// TIA Portal project "Kap_5_Uebung_Schutztuer_CPU_1500_V14_V15.1" (V15.1)

(* hardware
DEVICE "S71500/ET200MP-Station_1"  S7-1500 station
   slot 0: "Profilschiene_0"  6ES7 590-1***0-0AA0
   slot 1: "PLC_1"  CPU 1511-1 PN  6ES7 511-1AK01-0AB0  V1.8
   slot 2: "AI 8xU/I/RTD/TC ST_1"  AI 8xU/I/RTD/TC ST  6ES7 531-7KF00-0AB0  V2.0
   slot 3: "AI 8xU/I/RTD/TC ST_2"  AI 8xU/I/RTD/TC ST  6ES7 531-7KF00-0AB0  V2.0
   slot 4: "AI 8xU/I/RTD/TC ST_3"  AI 8xU/I/RTD/TC ST  6ES7 531-7KF00-0AB0  V2.0
   slot 5: "AI 8xU/I/RTD/TC ST_4"  AI 8xU/I/RTD/TC ST  6ES7 531-7KF00-0AB0  V2.0
   slot 6: "DI 16x24VDC BA_1"  DI 16x24VDC BA  6ES7 521-1BH10-0AA0  V1.0
*)

// ===== PLC "PLC_1"  CPU 1511-1 PN =====

VAR_GLOBAL   // PLC tag table "SchutzTuer"
   "SchutztuerGeschlossen_S1" AT %E0.0 : Bool;
   "SchutztuerGeschlossen_S2" AT %E0.1 : Bool;
   "SchutztuerGeoeffnet_S3" AT %E0.2 : Bool;
   "SchutztuerGeoeffnet_S4" AT %E0.3 : Bool;
   "FreigabeSignal" AT %A0.0 : Bool;
   "SchutztuerWarAuf" AT %M0.0 : Bool;
END_VAR

FUNCTION "MHJ-PLC-Lab-Function-S71500" : Void   // FC1, SCL
{ S7_Optimized_Access := 'TRUE' }
VERSION : 0.1
   VAR_TEMP
      Value : Byte;
      ForCounter : Int;
   END_VAR
   VAR CONSTANT
      Value_01_DW : DWord := 16#1223_5486;
      Value_02_DW : DWord := 16#A6C9_D1F5;
   END_VAR
BEGIN

   #Value:=PEEK(area := 16#82,
        dbNumber := 0,
        byteOffset := 511);
   #Value := #Value + 1;

   POKE(area := 16#82,
        dbNumber := 0,
        byteOffset := 511,
        value := #Value);

   POKE(area := 16#82,
        dbNumber := 0,
        byteOffset := 1016,
        value := #Value_01_DW);
   POKE(area := 16#82,
        dbNumber := 0,
        byteOffset := 1020,
        value := #Value_02_DW);
   FOR #ForCounter := 0 TO 63 DO
       #Value := PEEK(area := 16#1,
                      dbNumber := 0,
                      byteOffset := #ForCounter);
       POKE(area := 16#81,
            dbNumber := 0,
            byteOffset := #ForCounter,
            value := #Value);
   END_FOR;
   #Value := PEEK(area := 16#1,
                  dbNumber := 0,
                  byteOffset := 512);
   POKE(area := 16#82,
        dbNumber := 0,
        byteOffset := 512,
        value := #Value);
END_FUNCTION

ORGANIZATION_BLOCK "Main"   // OB1, FBD, ProgramCycle
TITLE = "Main Program Sweep (Cycle)"
{ S7_Optimized_Access := 'TRUE' }
VERSION : 0.1
   VAR_INPUT
      Initial_Call : Bool;   // Initial call of this OB
      Remanence : Bool;   // =True, if remanent data are available
   END_VAR
BEGIN

REGION Network 1
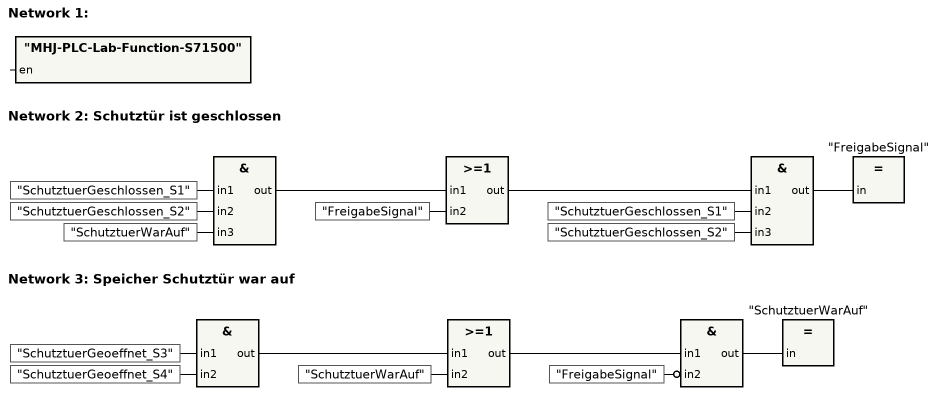
   "MHJ-PLC-Lab-Function-S71500"();
END_REGION

REGION Network 2: Schutztür ist geschlossen
   "FreigabeSignal" := (("SchutztuerGeschlossen_S1" AND "SchutztuerGeschlossen_S2" AND "SchutztuerWarAuf") OR "FreigabeSignal") AND "SchutztuerGeschlossen_S1" AND "SchutztuerGeschlossen_S2";
END_REGION

REGION Network 3: Speicher Schutztür war auf
   "SchutztuerWarAuf" := (("SchutztuerGeoeffnet_S3" AND "SchutztuerGeoeffnet_S4") OR "SchutztuerWarAuf") AND NOT "FreigabeSignal";
END_REGION
END_ORGANIZATION_BLOCK